// TIA Portal V16 export
// export: Created 2024-09-05T17:40:13.7608368Z, ExportSetting WithDefaults, DisplayName Totally Integrated Automation Portal, DisplayVersion V16 Update 6, DisplayName TIA Portal Version Control Interface, DisplayVersion V16 Update 2, DisplayName TIA Portal Openness, DisplayVersion V16 Update 6, DisplayName STEP 7 Professional, DisplayVersion V16 Update 6, DisplayName STEP 7 Safety, DisplayVersion V16, DisplayName WinCC Advanced, DisplayVersion V16 Update 6
TYPE "UDT_Slide"
// stored: IsFailsafeCompliant false
   STRUCT
      Enabled : Bool;
      FreeToInsert : Bool;
      PartInserted : Bool;
      SensorError : Bool;
      PartNotDetected : Bool;
   END_STRUCT;
END_TYPE
